TYPE ST_HMI_BASE_MODULE_OUT EXTENDS ST_HMI_BASE_CONTROL_OUT :
STRUCT
	stName				: ST_Text;
	stButtonNavigation	: ST_HMI_BUTTON_OUT;
	
	// info
	stState_Auto,
	stState_Home,
	stState				: ST_Text;	
	nStepChainName		: INT; // count visible rows from array aStepChainName
	aStepChainName		: ARRAY[0..CONST.iMaxIdxLocalStepChain] OF ST_Text;
	
	stManual			: ST_HMI_BASE_MODULE_MANUAL_OUT;
END_STRUCT
END_TYPE

(* stored: Version 1.1.0.1, ProductVersion 3.1.4024.12
   DUT ST_HMI_BASE_MODULE_OUT: Id {5dfdd26a-dbb1-4007-ac6f-059f6beda8be} *)
